FUNCTION_BLOCK Recipe_10055_Summerday
VAR_INPUT
	execute: BOOL;
	Order: DUT_RECIPEORDER;
END_VAR
VAR_OUTPUT
	RecipeInfo: DUT_RECIPEOFFER;
	RecipeDone: BOOL;
	InitDone: BOOL;
	Ready: BOOL;
END_VAR
VAR
	userparametersum: LREAL;
	StepDone: BOOL;
	i: INT;
	Command: ARRAY[1..5] OF DUT_RecipeCommand;
	NextSkill: BOOL;
	SectionReady: BOOL;
END_VAR

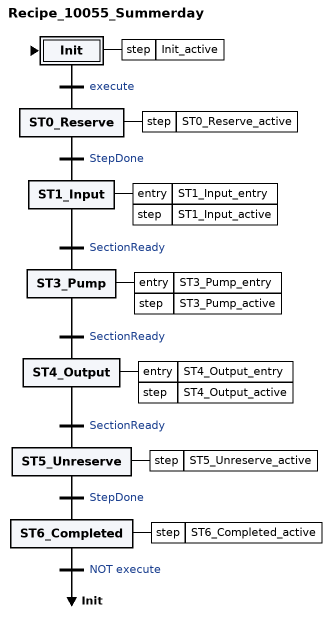
INITIAL_STEP Init:
    Init_active(N);  // step action
END_STEP
TRANSITION FROM Init TO ST0_Reserve
    := execute;
END_TRANSITION
STEP ST0_Reserve:
    ST0_Reserve_active(N);  // step action
END_STEP
TRANSITION FROM ST0_Reserve TO ST1_Input
    := StepDone;
END_TRANSITION
STEP ST1_Input:
    ST1_Input_entry(P1);  // entry action
    ST1_Input_active(N);  // step action
END_STEP
TRANSITION FROM ST1_Input TO ST3_Pump
    := SectionReady;
END_TRANSITION
STEP ST3_Pump:
    ST3_Pump_entry(P1);  // entry action
    ST3_Pump_active(N);  // step action
END_STEP
TRANSITION FROM ST3_Pump TO ST4_Output
    := SectionReady;
END_TRANSITION
STEP ST4_Output:
    ST4_Output_entry(P1);  // entry action
    ST4_Output_active(N);  // step action
END_STEP
TRANSITION FROM ST4_Output TO ST5_Unreserve
    := SectionReady;
END_TRANSITION
STEP ST5_Unreserve:
    ST5_Unreserve_active(N);  // step action
END_STEP
TRANSITION FROM ST5_Unreserve TO ST6_Completed
    := StepDone;
END_TRANSITION
STEP ST6_Completed:
    ST6_Completed_active(N);  // step action
END_STEP
TRANSITION FROM ST6_Completed TO Init
    := NOT execute;
END_TRANSITION

ACTION ST32a_DoseStart_active:
//RT: 2014.11.23: Summe aller zutaten zum Normiren

userparametersum := 0;
FOR i := 1 TO UserParameterCnt DO
	IF NOT (order.UserParameter[i].Value = 0) THEN
		userparametersum := userparametersum + order.UserParameter[i].Value;
	
	END_IF
END_FOR
IF userparametersum = 0 THEN
userparametersum := -1;
END_IF

//RT: 2014.11.23: Start wert des Arrays setzen
i := 1;
NextSkill := TRUE ;
END_ACTION

ACTION ST4_Output_active:
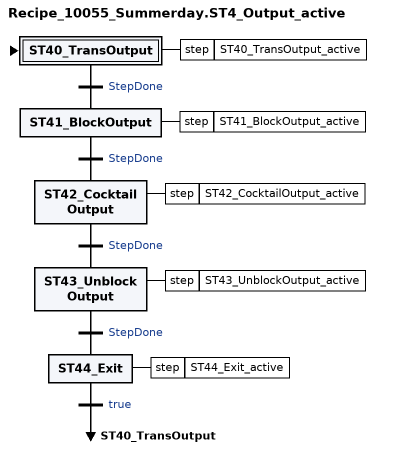
INITIAL_STEP ST40_TransOutput:
    ST40_TransOutput_active(N);  // step action
END_STEP
TRANSITION FROM ST40_TransOutput TO ST41_BlockOutput
    := StepDone;
END_TRANSITION
STEP ST41_BlockOutput:
    ST41_BlockOutput_active(N);  // step action
END_STEP
TRANSITION FROM ST41_BlockOutput TO ST42_CocktailOutput
    := StepDone;
END_TRANSITION
STEP ST42_CocktailOutput:
    ST42_CocktailOutput_active(N);  // step action
END_STEP
TRANSITION FROM ST42_CocktailOutput TO ST43_UnblockOutput
    := StepDone;
END_TRANSITION
STEP ST43_UnblockOutput:
    ST43_UnblockOutput_active(N);  // step action
END_STEP
TRANSITION FROM ST43_UnblockOutput TO ST44_Exit
    := StepDone;
END_TRANSITION
STEP ST44_Exit:
    ST44_Exit_active(N);  // step action
END_STEP
TRANSITION FROM ST44_Exit TO ST40_TransOutput
    := true;
END_TRANSITION
END_ACTION

ACTION Init_active:
//RT: 2014.11.23: Vorbereiten der daten und der HMI
RecipeDone := FALSE;

// Initialisation of Recipe Parameters an name etc
RecipeInfo.Name := 'Summerday';
RecipeInfo.Description := 'Flavoursome cocktail painting a picture of a beautiful summer day';
RecipeInfo.Dummy := FALSE;
RecipeInfo.RecipeID := 10055; 	// 
Initdone := TRUE;

//RT: 2014.11.23: wenn weniger als 5 alle lehren skills SkillID := 0
Command[1].SkillID := 1118;
Command[1].SkillName := 'Strawberry';
Command[1].Quantity := 14;

Command[2].SkillID := 1112;
Command[2].SkillName := 'Lemon Juice';
Command[2].Quantity := 14;

Command[3].SkillID := 1114;
Command[3].SkillName := 'Pineapple Juice';
Command[3].Quantity := 36;

Command[4].SkillID := 1117;
Command[4].SkillName := 'Orange Juice';
Command[4].Quantity := 36;

Command[5].SkillID := 0;
Command[5].SkillName := 'Nothing';
Command[5].Quantity := 0;








//Parameter 0:

	RecipeInfo.UserParameter[0].Dummy 		:= FALSE;
	RecipeInfo.UserParameter[0].Default		:= 200;
	RecipeInfo.UserParameter[0].Description	:= 'Gives the total fluid amount in the glass';
	RecipeInfo.UserParameter[0].MaxValue	:= 200;
	RecipeInfo.UserParameter[0].MinValue	:= 10;
	RecipeInfo.UserParameter[0].Name		:= 'Total Liquid Amount';
	RecipeInfo.UserParameter[0].Unit		:= 'ml';
	
//Parameter 1-5:
FOR i := 1 TO 5 DO
	IF Command[i].SkillID = 0 THEN
		RecipeInfo.UserParameter[i].Dummy 		:= TRUE;
	ELSE
		RecipeInfo.UserParameter[i].Dummy 		:= FALSE;
		RecipeInfo.UserParameter[i].Default		:= Command[i].Quantity;
		RecipeInfo.UserParameter[i].Description	:= Command[i].SkillName;
		RecipeInfo.UserParameter[i].MaxValue	:= 100;
		RecipeInfo.UserParameter[i].MinValue	:= 1;
		RecipeInfo.UserParameter[i].Name		:= Command[i].SkillName;
		RecipeInfo.UserParameter[i].Unit		:= 'ml';	
	END_IF
END_FOR
END_ACTION

ACTION ST44_Exit_active:
SectionReady := TRUE;
END_ACTION

ACTION ST34_Exit_active:
SectionReady := TRUE;
END_ACTION

ACTION ST13_UnblockInput_active:
//RT: 2014.11.23: Gibt Mover Position Frei
StepDone := FALSE;

//Skill auswählen
ExecuteSkill.SkillID 		:= 1316;
ExecuteSkill.SkillName	 	:= 'Unblock';

//Parameter setzen

ExecuteSkill.Parameter[1].ID := 1;
ExecuteSkill.Parameter[1].Name := 'TaskID';
ExecuteSkill.Parameter[1].Value := Order.TaskID;


(*
ExecuteSkill.Parameter[2].ID := ;
ExecuteSkill.Parameter[2].Name := '';
ExecuteSkill.Parameter[2].Value := ;
*)

(*
ExecuteSkill.Parameter[3].ID := ;
ExecuteSkill.Parameter[3].Name := '';
ExecuteSkill.Parameter[3].Value := ;
*)

(*
ExecuteSkill.Parameter[4].ID := ;
ExecuteSkill.Parameter[4].Name := '';
ExecuteSkill.Parameter[4].Value := ;
*)

(*
ExecuteSkill.Parameter[5].ID := ;
ExecuteSkill.Parameter[5].Name := '';
ExecuteSkill.Parameter[5].Value := ;
*)



ExecuteSkill();

StepDone := ExecuteSkill.Done;
END_ACTION

ACTION ST32b_Dose_exit:

END_ACTION

ACTION ST1_Input_entry:
SectionReady := FALSE;
END_ACTION

ACTION ST3_Pump_entry:
SectionReady := FALSE;
END_ACTION

ACTION ST31_BlockPump_active:
//RT: 2014.11.23: Blockirt den Mover an Position
StepDone := FALSE;

//Skill auswählen
ExecuteSkill.SkillID 		:= 1315;
ExecuteSkill.SkillName	 	:= 'Block';

//Parameter setzen

ExecuteSkill.Parameter[1].ID := 1;
ExecuteSkill.Parameter[1].Name := 'TaskID';
ExecuteSkill.Parameter[1].Value := Order.TaskID;


(*
ExecuteSkill.Parameter[2].ID := ;
ExecuteSkill.Parameter[2].Name := '';
ExecuteSkill.Parameter[2].Value := ;
*)

(*
ExecuteSkill.Parameter[3].ID := ;
ExecuteSkill.Parameter[3].Name := '';
ExecuteSkill.Parameter[3].Value := ;
*)

(*
ExecuteSkill.Parameter[4].ID := ;
ExecuteSkill.Parameter[4].Name := '';
ExecuteSkill.Parameter[4].Value := ;
*)

(*
ExecuteSkill.Parameter[5].ID := ;
ExecuteSkill.Parameter[5].Name := '';
ExecuteSkill.Parameter[5].Value := ;
*)



ExecuteSkill();

StepDone := ExecuteSkill.Done;
END_ACTION

ACTION ST1_Input_active:
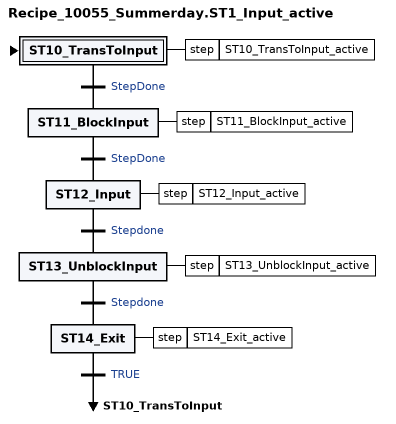
INITIAL_STEP ST10_TransToInput:
    ST10_TransToInput_active(N);  // step action
END_STEP
TRANSITION FROM ST10_TransToInput TO ST11_BlockInput
    := StepDone;
END_TRANSITION
STEP ST11_BlockInput:
    ST11_BlockInput_active(N);  // step action
END_STEP
TRANSITION FROM ST11_BlockInput TO ST12_Input
    := StepDone;
END_TRANSITION
STEP ST12_Input:
    ST12_Input_active(N);  // step action
END_STEP
TRANSITION FROM ST12_Input TO ST13_UnblockInput
    := Stepdone;
END_TRANSITION
STEP ST13_UnblockInput:
    ST13_UnblockInput_active(N);  // step action
END_STEP
TRANSITION FROM ST13_UnblockInput TO ST14_Exit
    := Stepdone;
END_TRANSITION
STEP ST14_Exit:
    ST14_Exit_active(N);  // step action
END_STEP
TRANSITION FROM ST14_Exit TO ST10_TransToInput
    := TRUE;
END_TRANSITION
END_ACTION

ACTION ST32b_Dose_active:
//RT: 2014.11.23: Die Dosir Skills anlegen
StepDone := FALSE;

//Skill auswählen
ExecuteSkill.SkillID 		:= Command[i].SkillID;
ExecuteSkill.SkillName	 	:= Command[i].SkillName;
//Parameter setzen

ExecuteSkill.Parameter[0].ID := 1;
ExecuteSkill.Parameter[0].Name := 'Quantity';
//order.userParameter[0] = amount
ExecuteSkill.Parameter[0].Value := order.UserParameter[0].Value * order.UserParameter[i].Value / userparametersum ;//Summe aller Zutatenmengen;

(*
ExecuteSkill.Parameter[2].ID := ;
ExecuteSkill.Parameter[2].Name := '';
ExecuteSkill.Parameter[2].Value := ;
*)

(*
ExecuteSkill.Parameter[3].ID := ;
ExecuteSkill.Parameter[3].Name := '';
ExecuteSkill.Parameter[3].Value := ;
*)

(*
ExecuteSkill.Parameter[4].ID := ;
ExecuteSkill.Parameter[4].Name := '';
ExecuteSkill.Parameter[4].Value := ;
*)

(*
ExecuteSkill.Parameter[5].ID := ;
ExecuteSkill.Parameter[5].Name := '';
ExecuteSkill.Parameter[5].Value := ;
*)


ExecuteSkill();

StepDone := ExecuteSkill.Done;

i := i + 1 ;

IF i = 6 THEN
	NextSkill := FALSE;
ELSIF Command[i].SkillID = 0 THEN
	NextSkill := FALSE;
ELSE
	NextSkill := TRUE;
END_IF
END_ACTION

ACTION ST0_Reserve_active:
//RT: 2014.11.23: Reservire einen Mover

StepDone := FALSE;
RecipeDone := FALSE;
//Skill auswählen
ExecuteSkill.SkillID 		:= 1310;
ExecuteSkill.SkillName	 	:= 'Reserve';

//Parameter setzen

ExecuteSkill.Parameter[1].ID := 1;
ExecuteSkill.Parameter[1].Name := 'TaskID';
ExecuteSkill.Parameter[1].Value := Order.TaskID;

(*
ExecuteSkill.Parameter[2].ID := ;
ExecuteSkill.Parameter[2].Name := '';
ExecuteSkill.Parameter[2].Value := ;
*)

(*
ExecuteSkill.Parameter[3].ID := ;
ExecuteSkill.Parameter[3].Name := '';
ExecuteSkill.Parameter[3].Value := ;
*)

(*
ExecuteSkill.Parameter[4].ID := ;
ExecuteSkill.Parameter[4].Name := '';
ExecuteSkill.Parameter[4].Value := ;
*)

(*
ExecuteSkill.Parameter[5].ID := ;
ExecuteSkill.Parameter[5].Name := '';
ExecuteSkill.Parameter[5].Value := ;
*)

ExecuteSkill();

StepDone := ExecuteSkill.Done;
END_ACTION

ACTION ST14_Exit_active:
SectionReady := TRUE;
END_ACTION

ACTION ST12_Input_active:
//RT: 2014.11.23: Input Modul auslösen
StepDone := FALSE;

//Skill auswählen
ExecuteSkill.SkillID 		:= 1402;
ExecuteSkill.SkillName	 	:= 'Input';

//Parameter setzen

ExecuteSkill.Parameter[1].ID := 1;
ExecuteSkill.Parameter[1].Name := 'TaskID';
ExecuteSkill.Parameter[1].Value := Order.TaskID;


(*
ExecuteSkill.Parameter[2].ID := ;
ExecuteSkill.Parameter[2].Name := '';
ExecuteSkill.Parameter[2].Value := ;
*)

(*
ExecuteSkill.Parameter[3].ID := ;
ExecuteSkill.Parameter[3].Name := '';
ExecuteSkill.Parameter[3].Value := ;
*)

(*
ExecuteSkill.Parameter[4].ID := ;
ExecuteSkill.Parameter[4].Name := '';
ExecuteSkill.Parameter[4].Value := ;
*)

(*
ExecuteSkill.Parameter[5].ID := ;
ExecuteSkill.Parameter[5].Name := '';
ExecuteSkill.Parameter[5].Value := ;
*)



ExecuteSkill();

StepDone := ExecuteSkill.Done;
END_ACTION

ACTION ST33_UnblockPump_active:
//RT: 2014.11.23: Gibt Mover Position Frei
StepDone := FALSE;

//Skill auswählen
ExecuteSkill.SkillID 		:= 1316;
ExecuteSkill.SkillName	 	:= 'Unblock';

//Parameter setzen

ExecuteSkill.Parameter[1].ID := 1;
ExecuteSkill.Parameter[1].Name := 'TaskID';
ExecuteSkill.Parameter[1].Value := Order.TaskID;


(*
ExecuteSkill.Parameter[2].ID := ;
ExecuteSkill.Parameter[2].Name := '';
ExecuteSkill.Parameter[2].Value := ;
*)

(*
ExecuteSkill.Parameter[3].ID := ;
ExecuteSkill.Parameter[3].Name := '';
ExecuteSkill.Parameter[3].Value := ;
*)

(*
ExecuteSkill.Parameter[4].ID := ;
ExecuteSkill.Parameter[4].Name := '';
ExecuteSkill.Parameter[4].Value := ;
*)

(*
ExecuteSkill.Parameter[5].ID := ;
ExecuteSkill.Parameter[5].Name := '';
ExecuteSkill.Parameter[5].Value := ;
*)



ExecuteSkill();

StepDone := ExecuteSkill.Done;
END_ACTION

ACTION ST1_Reserve0_active:
//RT: 2014.11.23: Reservire einen Mover

StepDone := FALSE;
RecipeDone := FALSE;
//Skill auswählen
ExecuteSkill.SkillID 		:= 1310;
ExecuteSkill.SkillName	 	:= 'Reserve';

//Parameter setzen

ExecuteSkill.Parameter[1].ID := 1;
ExecuteSkill.Parameter[1].Name := 'TaskID';
ExecuteSkill.Parameter[1].Value := Order.TaskID;

(*
ExecuteSkill.Parameter[2].ID := ;
ExecuteSkill.Parameter[2].Name := '';
ExecuteSkill.Parameter[2].Value := ;
*)

(*
ExecuteSkill.Parameter[3].ID := ;
ExecuteSkill.Parameter[3].Name := '';
ExecuteSkill.Parameter[3].Value := ;
*)

(*
ExecuteSkill.Parameter[4].ID := ;
ExecuteSkill.Parameter[4].Name := '';
ExecuteSkill.Parameter[4].Value := ;
*)

(*
ExecuteSkill.Parameter[5].ID := ;
ExecuteSkill.Parameter[5].Name := '';
ExecuteSkill.Parameter[5].Value := ;
*)

ExecuteSkill();

StepDone := ExecuteSkill.Done;
END_ACTION

ACTION ST42_CocktailOutput_active:
//RT: 2014.11.23: Ausgeben des Produktes
StepDone := FALSE;

//Skill auswählen
ExecuteSkill.SkillID 		:= 1403;
ExecuteSkill.SkillName	 	:= 'Output';

//Parameter setzen

ExecuteSkill.Parameter[1].ID := 1;
ExecuteSkill.Parameter[1].Name := 'TaskID';
ExecuteSkill.Parameter[1].Value := Order.TaskID;


(*
ExecuteSkill.Parameter[2].ID := ;
ExecuteSkill.Parameter[2].Name := '';
ExecuteSkill.Parameter[2].Value := ;
*)

(*
ExecuteSkill.Parameter[3].ID := ;
ExecuteSkill.Parameter[3].Name := '';
ExecuteSkill.Parameter[3].Value := ;
*)

(*
ExecuteSkill.Parameter[4].ID := ;
ExecuteSkill.Parameter[4].Name := '';
ExecuteSkill.Parameter[4].Value := ;
*)

(*
ExecuteSkill.Parameter[5].ID := ;
ExecuteSkill.Parameter[5].Name := '';
ExecuteSkill.Parameter[5].Value := ;
*)



ExecuteSkill();

StepDone := ExecuteSkill.Done;
END_ACTION

ACTION ST11_BlockInput_active:
//RT: 2014.11.23: Blockirt den Mover an Position
StepDone := FALSE;

//Skill auswählen
ExecuteSkill.SkillID 		:= 1315;
ExecuteSkill.SkillName	 	:= 'Block';

//Parameter setzen

ExecuteSkill.Parameter[1].ID := 1;
ExecuteSkill.Parameter[1].Name := 'TaskID';
ExecuteSkill.Parameter[1].Value := Order.TaskID;


(*
ExecuteSkill.Parameter[2].ID := ;
ExecuteSkill.Parameter[2].Name := '';
ExecuteSkill.Parameter[2].Value := ;
*)

(*
ExecuteSkill.Parameter[3].ID := ;
ExecuteSkill.Parameter[3].Name := '';
ExecuteSkill.Parameter[3].Value := ;
*)

(*
ExecuteSkill.Parameter[4].ID := ;
ExecuteSkill.Parameter[4].Name := '';
ExecuteSkill.Parameter[4].Value := ;
*)

(*
ExecuteSkill.Parameter[5].ID := ;
ExecuteSkill.Parameter[5].Name := '';
ExecuteSkill.Parameter[5].Value := ;
*)



ExecuteSkill();

StepDone := ExecuteSkill.Done;
END_ACTION

ACTION ST10_TransToInput_active:
//RT: 2014.11.23: Mover zum Input

StepDone := FALSE;

//Skill auswählen
ExecuteSkill.SkillID 		:= 1320;
ExecuteSkill.SkillName	 	:= 'Transport';

//Parameter setzen

ExecuteSkill.Parameter[3].ID := 3;
ExecuteSkill.Parameter[3].Name := 'Velocity';
ExecuteSkill.Parameter[3].Value := 1000;



ExecuteSkill.Parameter[1].ID :=  1;
ExecuteSkill.Parameter[1].Name := 'TargetPosition X';
ExecuteSkill.Parameter[1].Value := 30 ;
ExecuteSkill.Parameter[1].StringValue := '#DP#2#XPosition';



ExecuteSkill.Parameter[2].ID := 2;
ExecuteSkill.Parameter[2].Name := 'TargetPosition Z';
ExecuteSkill.Parameter[2].Value := 100;// ZCookieModule - ZCookieModuleCalibration - 2* Cookiethickness + toppingthickness+ Preasureheight  ;



(*
ExecuteSkill.Parameter[4].ID := 4;
ExecuteSkill.Parameter[4].Name := 'Acceleration';
ExecuteSkill.Parameter[4].Value := 0 ;
*)

(*
ExecuteSkill.Parameter[5].ID := ;
ExecuteSkill.Parameter[5].Name := '';
ExecuteSkill.Parameter[5].Value := ;
*)



ExecuteSkill();

StepDone := ExecuteSkill.Done;
END_ACTION

ACTION ST30_TransPump_active:
//RT: 2014.11.23: Mover zum Pump
StepDone := FALSE;

//Skill auswählen
ExecuteSkill.SkillID 		:= 1320;
ExecuteSkill.SkillName	 	:= 'Transport';

//Parameter setzen

ExecuteSkill.Parameter[3].ID := 3;
ExecuteSkill.Parameter[3].Name := 'Velocity';
ExecuteSkill.Parameter[3].Value := 1000;



ExecuteSkill.Parameter[1].ID :=  1;
ExecuteSkill.Parameter[1].Name := 'TargetPosition X';
ExecuteSkill.Parameter[1].Value := 30 ;
ExecuteSkill.Parameter[1].StringValue := '#DP#2#XPosition';



ExecuteSkill.Parameter[2].ID := 2;
ExecuteSkill.Parameter[2].Name := 'TargetPosition Z';
ExecuteSkill.Parameter[2].Value := 20;// ZCookieModule - ZCookieModuleCalibration - 2* Cookiethickness + toppingthickness+ Preasureheight  ;



(*
ExecuteSkill.Parameter[4].ID := 4;
ExecuteSkill.Parameter[4].Name := 'Acceleration';
ExecuteSkill.Parameter[4].Value := 0 ;
*)

(*
ExecuteSkill.Parameter[5].ID := ;
ExecuteSkill.Parameter[5].Name := '';
ExecuteSkill.Parameter[5].Value := ;
*)



ExecuteSkill();

StepDone := ExecuteSkill.Done;
END_ACTION

ACTION ST6_Completed_active:
//RT: 2014.11.23: Warte auf Execute = False
RecipeDone := TRUE;
StepDone := FALSE;
END_ACTION

ACTION ST5_Unreserve_active:
//RT: 2014.11.23: Mover Freigeben
StepDone := FALSE;

//Skill auswählen
ExecuteSkill.SkillID 		:= 1311;
ExecuteSkill.SkillName	 	:= 'Unreserve';

//Parameter setzen

ExecuteSkill.Parameter[1].ID := 1;
ExecuteSkill.Parameter[1].Name := 'TaskID';
ExecuteSkill.Parameter[1].Value := Order.TaskID;


(*
ExecuteSkill.Parameter[2].ID := ;
ExecuteSkill.Parameter[2].Name := '';
ExecuteSkill.Parameter[2].Val ue := ;
*)

(*
ExecuteSkill.Parameter[3].ID := ;
ExecuteSkill.Parameter[3].Name := '';
ExecuteSkill.Parameter[3].Value := ;
*)

(*
ExecuteSkill.Parameter[4].ID := ;
ExecuteSkill.Parameter[4].Name := '';
ExecuteSkill.Parameter[4].Value := ;
*)

(*
ExecuteSkill.Parameter[5].ID := ;
ExecuteSkill.Parameter[5].Name := '';
ExecuteSkill.Parameter[5].Value := ;
*)



ExecuteSkill();

StepDone := ExecuteSkill.Done;
END_ACTION

ACTION ST40_TransOutput_active:
//RT: 2014.11.23: Mover zum Output
StepDone := FALSE;

//Skill auswählen
ExecuteSkill.SkillID 		:= 1320;
ExecuteSkill.SkillName	 	:= 'Transport';

//Parameter setzen

ExecuteSkill.Parameter[3].ID := 3;
ExecuteSkill.Parameter[3].Name := 'Velocity';
ExecuteSkill.Parameter[3].Value := 300;



ExecuteSkill.Parameter[1].ID :=  1;
ExecuteSkill.Parameter[1].Name := 'TargetPosition X';
ExecuteSkill.Parameter[1].Value := 30 ;
ExecuteSkill.Parameter[1].StringValue := '#DP#2#XPosition';



ExecuteSkill.Parameter[2].ID := 2;
ExecuteSkill.Parameter[2].Name := 'TargetPosition Z';
ExecuteSkill.Parameter[2].Value := ZInputOutput;// ZCookieModule - ZCookieModuleCalibration - 2* Cookiethickness + toppingthickness+ Preasureheight  ;



(* ExecuteSkill.Parameter[4].ID := 4;
ExecuteSkill.Parameter[4].Name := 'Acceleration';
ExecuteSkill.Parameter[4].Value :=0 ;

*)
(*
ExecuteSkill.Parameter[5].ID := ;
ExecuteSkill.Parameter[5].Name := '';
ExecuteSkill.Parameter[5].Value := ;
*)



ExecuteSkill();

StepDone := ExecuteSkill.Done;
END_ACTION

ACTION ST43_UnblockOutput_active:
//RT: 2014.11.23: Gibt Mover Position Frei
StepDone := FALSE;

//Skill auswählen
ExecuteSkill.SkillID 		:= 1316;
ExecuteSkill.SkillName	 	:= 'Unblock';

//Parameter setzen

ExecuteSkill.Parameter[1].ID := 1;
ExecuteSkill.Parameter[1].Name := 'TaskID';
ExecuteSkill.Parameter[1].Value := Order.TaskID;


(*
ExecuteSkill.Parameter[2].ID := ;
ExecuteSkill.Parameter[2].Name := '';
ExecuteSkill.Parameter[2].Value := ;
*)

(*
ExecuteSkill.Parameter[3].ID := ;
ExecuteSkill.Parameter[3].Name := '';
ExecuteSkill.Parameter[3].Value := ;
*)

(*
ExecuteSkill.Parameter[4].ID := ;
ExecuteSkill.Parameter[4].Name := '';
ExecuteSkill.Parameter[4].Value := ;
*)

(*
ExecuteSkill.Parameter[5].ID := ;
ExecuteSkill.Parameter[5].Name := '';
ExecuteSkill.Parameter[5].Value := ;
*)



ExecuteSkill();

StepDone := ExecuteSkill.Done;
END_ACTION

ACTION ST4_Output_entry:
SectionReady := FALSE;
END_ACTION

ACTION ST3_Pump_active:
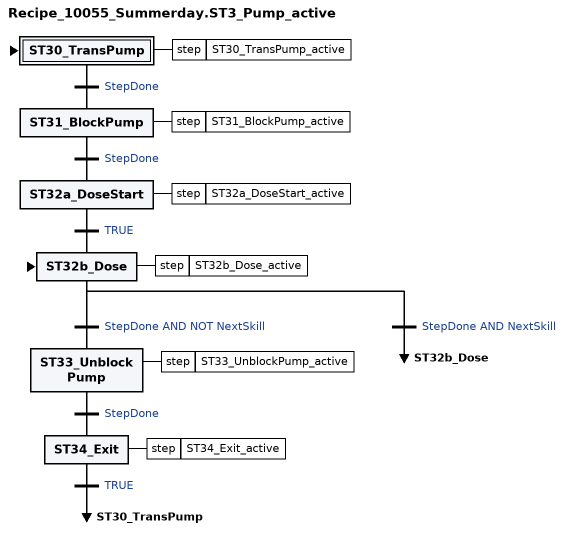
INITIAL_STEP ST30_TransPump:
    ST30_TransPump_active(N);  // step action
END_STEP
TRANSITION FROM ST30_TransPump TO ST31_BlockPump
    := StepDone;
END_TRANSITION
STEP ST31_BlockPump:
    ST31_BlockPump_active(N);  // step action
END_STEP
TRANSITION FROM ST31_BlockPump TO ST32a_DoseStart
    := StepDone;
END_TRANSITION
STEP ST32a_DoseStart:
    ST32a_DoseStart_active(N);  // step action
END_STEP
TRANSITION FROM ST32a_DoseStart TO ST32b_Dose
    := TRUE;
END_TRANSITION
STEP ST32b_Dose:
    ST32b_Dose_active(N);  // step action
END_STEP
TRANSITION FROM ST32b_Dose TO ST33_UnblockPump
    := StepDone AND NOT NextSkill;
END_TRANSITION
STEP ST33_UnblockPump:
    ST33_UnblockPump_active(N);  // step action
END_STEP
TRANSITION FROM ST33_UnblockPump TO ST34_Exit
    := StepDone;
END_TRANSITION
STEP ST34_Exit:
    ST34_Exit_active(N);  // step action
END_STEP
TRANSITION FROM ST34_Exit TO ST30_TransPump
    := TRUE;
END_TRANSITION
TRANSITION FROM ST32b_Dose TO ST32b_Dose
    := StepDone AND NextSkill;
END_TRANSITION
END_ACTION

ACTION ST41_BlockOutput_active:
//RT: 2014.11.23: Blockirt den Mover an Position
StepDone := FALSE;

//Skill auswählen
ExecuteSkill.SkillID 		:= 1315;
ExecuteSkill.SkillName	 	:= 'Block';

//Parameter setzen

ExecuteSkill.Parameter[1].ID := 1;
ExecuteSkill.Parameter[1].Name := 'TaskID';
ExecuteSkill.Parameter[1].Value := Order.TaskID;


(*
ExecuteSkill.Parameter[2].ID := ;
ExecuteSkill.Parameter[2].Name := '';
ExecuteSkill.Parameter[2].Value := ;
*)

(*
ExecuteSkill.Parameter[3].ID := ;
ExecuteSkill.Parameter[3].Name := '';
ExecuteSkill.Parameter[3].Value := ;
*)

(*
ExecuteSkill.Parameter[4].ID := ;
ExecuteSkill.Parameter[4].Name := '';
ExecuteSkill.Parameter[4].Value := ;
*)

(*
ExecuteSkill.Parameter[5].ID := ;
ExecuteSkill.Parameter[5].Name := '';
ExecuteSkill.Parameter[5].Value := ;
*)



ExecuteSkill();

StepDone := ExecuteSkill.Done;
END_ACTION

END_FUNCTION_BLOCK

(* stored: Version 1.1.0.1, ProductVersion 3.1.0.25
   POU Recipe_10055_Summerday: Id {82a675fc-fc85-412c-a9a9-47d52c8a98ae}
   Action ST32a_DoseStart_active: Id {00cc2ec7-fd28-4715-9a5c-2ede9048d040}
   Action ST4_Output_active: Id {0f717800-08e9-4b56-88a5-e045d87d84ea}
   Action Init_active: Id {13ac6fe6-06a9-404a-b81f-0eec9c79124a}
   Action ST44_Exit_active: Id {1c264647-e14a-4a6e-a486-135b2468b235}
   Action ST34_Exit_active: Id {23d18f10-34a5-43cd-a280-aa65f47e87a5}
   Action ST13_UnblockInput_active: Id {2d892164-3930-4ab0-8be1-fa38bf122d7b}
   Action ST32b_Dose_exit: Id {2f9c3337-4860-4acf-a0ac-5f63f51eea15}
   Action ST1_Input_entry: Id {3b3872a1-235e-4ac3-bac3-99e6b00ce136}
   Action ST3_Pump_entry: Id {43008316-2bbd-4739-a100-4ffb22433397}
   Action ST31_BlockPump_active: Id {4e66ed96-0e56-4cea-86ad-1972807bf2ea}
   Action ST1_Input_active: Id {5fc6ccb9-8c23-4767-a3ae-78d383d78bfa}
   Action ST32b_Dose_active: Id {a3e360c4-3ffc-46da-a602-e50fd3fb4f2a}
   Action ST0_Reserve_active: Id {a504f1ed-1f32-4191-b6a4-8253d22d5d43}
   Action ST14_Exit_active: Id {a7afd5fa-689b-4fe4-b7d1-b6846f8351f5}
   Action ST12_Input_active: Id {aa84b100-b4d3-497a-aa6e-75a45d87b539}
   Action ST33_UnblockPump_active: Id {ac21e5e8-d0ce-4c51-8902-4f6f8d61ccbb}
   Action ST1_Reserve0_active: Id {ac5c1404-e3ce-42bd-bbbf-a1cb05f3128c}
   Action ST42_CocktailOutput_active: Id {b3cb0689-1538-479d-aca4-f3368e43f154}
   Action ST11_BlockInput_active: Id {b5f091b4-9506-4d2e-9b82-3f8d8a1481ad}
   Action ST10_TransToInput_active: Id {bf986d65-18fc-49cd-816b-726980b112cf}
   Action ST30_TransPump_active: Id {bfe09705-e14f-4b89-b567-a8b7c1626aa8}
   Action ST6_Completed_active: Id {c38683f7-42ab-4714-8f65-994a93d0ff7a}
   Action ST5_Unreserve_active: Id {d532c0f7-7922-428c-a4af-27ab7ec6ec48}
   Action ST40_TransOutput_active: Id {dd8c28b1-f3e2-488f-bd84-d5d90b4fd192}
   Action ST43_UnblockOutput_active: Id {de2cda1c-68c1-4fd4-ba5f-a5f12feac9c3}
   Action ST4_Output_entry: Id {e7622d9d-7e84-4021-96f5-36cf91ffdfb1}
   Action ST3_Pump_active: Id {f6350d93-7487-4299-a660-e6186e40b465}
   Action ST41_BlockOutput_active: Id {f8160b39-4260-47f5-9e5c-96c7fba1e77d} *)
